Fanuc KAREL source: NC0030.KL

-- PROVISIONAL review KL for V940-1; original PC SHA256 17421e0115ae06eb4551ab419e4b332e2ef42d31b7094077018fdf0aaf0534d4
-- Incomplete behavior may be omitted. Consult companion uncertainty JSON. Do not deploy.
PROGRAM NC0030
%NOLOCKGROUP
-- UNRESOLVED_LOCAL_POOL 1 cells at code offset 3; source declarations unknown
-- DIRECT_LOCAL_WORD_ACCESS alone does not prove INTEGER, REAL, or BOOLEAN
BEGIN
  -- UNRESOLVED_PC offsets 0-8; opcodes 2B,2C,7B
  -- UNRESOLVED_PC offsets 13-20; opcodes 9D,23
  -- UNRESOLVED_PC offsets 25-42; opcodes 21,40,41,42
  -- UNRESOLVED_PC offsets 47-64; opcodes 21,40,41,42
  -- UNRESOLVED_PC offsets 69-86; opcodes 21,40,41,42
  -- UNRESOLVED_PC offsets 91-108; opcodes 21,40,41,42
  -- UNRESOLVED_PC offsets 113-130; opcodes 21,40,41,42
  -- UNRESOLVED_PC offsets 135-152; opcodes 21,40,41,42
  -- UNRESOLVED_PC offsets 157-174; opcodes 21,40,41,42
  -- UNRESOLVED_PC offsets 179-196; opcodes 21,40,41,42
  -- UNRESOLVED_PC offsets 201-218; opcodes 21,40,41,42
  -- UNRESOLVED_PC offsets 223-240; opcodes 21,40,41,42
  -- UNRESOLVED_PC offsets 245-262; opcodes 21,40,41,42
  -- UNRESOLVED_PC offsets 267-284; opcodes 21,40,41,42
  -- UNRESOLVED_PC offsets 289-306; opcodes 21,40,41,42
  -- UNRESOLVED_PC offsets 311-328; opcodes 21,40,41,42
  -- UNRESOLVED_PC offsets 333-350; opcodes 21,40,41,42
  -- UNRESOLVED_PC offsets 355-372; opcodes 21,40,41,42
  -- UNRESOLVED_PC offsets 377-394; opcodes 21,40,41,42
  -- UNRESOLVED_PC offsets 399-416; opcodes 21,40,41,42
  -- UNRESOLVED_PC offsets 421-451; opcodes 21,9D,52,23,7A,40,41,42
  -- UNRESOLVED_PC offsets 456-480; opcodes 21,2E,52,23,7A,43
  -- UNRESOLVED_PC offsets 485-503; opcodes 21,2E,52,23
  -- UNRESOLVED_PC offsets 508-524; opcodes 7A,40,41,42
  -- UNRESOLVED_PC offsets 529-553; opcodes 21,2E,52,23,7A,43
  -- UNRESOLVED_PC offsets 558-576; opcodes 21,2E,52,23
  -- UNRESOLVED_PC offsets 581-597; opcodes 7A,40,41,42
  -- UNRESOLVED_PC offsets 602-626; opcodes 21,2E,52,23,7A,43
  -- UNRESOLVED_PC offsets 631-649; opcodes 21,2E,52,23
  -- UNRESOLVED_PC offsets 654-670; opcodes 7A,40,41,42
  -- UNRESOLVED_PC offsets 675-699; opcodes 21,2E,52,23,7A,43
  -- UNRESOLVED_PC offsets 704-722; opcodes 21,2E,52,23
  -- UNRESOLVED_PC offsets 727-743; opcodes 7A,40,41,42
  -- UNRESOLVED_PC offsets 748-772; opcodes 21,2E,52,23,7A,43
  -- UNRESOLVED_PC offsets 777-795; opcodes 21,2E,52,23
  -- UNRESOLVED_PC offsets 800-816; opcodes 7A,40,41,42
  -- UNRESOLVED_PC offsets 821-845; opcodes 21,2E,52,23,7A,43
  -- UNRESOLVED_PC offsets 850-868; opcodes 21,2E,52,23
  -- UNRESOLVED_PC offsets 873-889; opcodes 7A,40,41,42
  -- UNRESOLVED_PC offsets 894-918; opcodes 21,2E,52,23,7A,43
  -- UNRESOLVED_PC offsets 923-941; opcodes 21,2E,52,23
  -- UNRESOLVED_PC offsets 946-962; opcodes 7A,40,41,42
  -- UNRESOLVED_PC offsets 967-991; opcodes 21,2E,52,23,7A,43
  -- UNRESOLVED_PC offsets 996-1014; opcodes 21,2E,52,23
  -- UNRESOLVED_PC offsets 1019-1035; opcodes 7A,40,41,42
  -- UNRESOLVED_PC offsets 1040-1064; opcodes 21,2E,52,23,7A,43
  -- UNRESOLVED_PC offsets 1069-1087; opcodes 21,2E,52,23
  -- UNRESOLVED_PC offsets 1092-1108; opcodes 7A,40,41,42
  -- UNRESOLVED_PC offsets 1113-1137; opcodes 21,2E,52,23,7A,43
  -- UNRESOLVED_PC offsets 1142-1160; opcodes 21,2E,52,23
  -- UNRESOLVED_PC offsets 1165-1181; opcodes 7A,40,41,42
  -- UNRESOLVED_PC offsets 1186-1210; opcodes 21,2E,52,23,7A,43
  -- UNRESOLVED_PC offsets 1215-1233; opcodes 21,2E,52,23
  -- UNRESOLVED_PC offsets 1238-1254; opcodes 7A,40,41,42
  -- UNRESOLVED_PC offsets 1259-1283; opcodes 21,2E,52,23,7A,43
  -- UNRESOLVED_PC offsets 1288-1306; opcodes 21,2E,52,23
  -- UNRESOLVED_PC offsets 1311-1327; opcodes 7A,40,41,42
  -- UNRESOLVED_PC offsets 1332-1356; opcodes 21,2E,52,23,7A,43
  -- UNRESOLVED_PC offsets 1361-1379; opcodes 21,2E,52,23
  -- UNRESOLVED_PC offsets 1384-1400; opcodes 7A,40,41,42
  -- UNRESOLVED_PC offsets 1405-1429; opcodes 21,2E,52,23,7A,43
  -- UNRESOLVED_PC offsets 1434-1452; opcodes 21,2E,52,23
  -- UNRESOLVED_PC offsets 1457-1473; opcodes 7A,40,41,42
  -- UNRESOLVED_PC offsets 1478-1502; opcodes 21,2E,52,23,7A,43
  -- UNRESOLVED_PC offsets 1507-1525; opcodes 21,2E,52,23
  -- UNRESOLVED_PC offsets 1530-1546; opcodes 7A,40,41,42
  -- UNRESOLVED_PC offsets 1551-1575; opcodes 21,2E,52,23,7A,43
  -- UNRESOLVED_PC offsets 1580-1598; opcodes 21,2E,52,23
  -- UNRESOLVED_PC offsets 1603-1619; opcodes 7A,40,41,42
  -- UNRESOLVED_PC offsets 1624-1648; opcodes 21,2E,52,23,7A,43
  -- UNRESOLVED_PC offsets 1653-1671; opcodes 21,2E,52,23
  -- UNRESOLVED_PC offsets 1676-1692; opcodes 7A,40,41,42
  -- UNRESOLVED_PC offsets 1697-1721; opcodes 21,2E,52,23,7A,43
  -- UNRESOLVED_PC offsets 1726-1744; opcodes 21,2E,52,23
  -- UNRESOLVED_PC offsets 1754-1758; opcodes 7F
  -- UNRESOLVED_PC offsets 1763-1767; opcodes 27,AA
  -- UNRESOLVED_PC offsets 1772-1776; opcodes 7F
END NC0030
